// TIA Portal project "TankMixer3" (V17)

(* hardware
DEVICE "S7-1500/ET200MP station_1"  S7-1500 station
   slot 0: "Rail_0"  Rack  6ES7 590-1***0-0AA0
   slot 1: "PLC_1"  CPU 1512C-1 PN  6ES7 512-1CK00-0AB0  V2.9
      slot 3: "CPU display_1"  6ES7591-1AA00-0AA0
      slot 32768: "PROFINET interface_1"  X1
         slot 32769: "Port_1"  X1 P1
         slot 32770: "Port_2"  X1 P2
      slot 34817: "Virtual CP interface port_1"  Virtual CP interface port  Virtual CP interface port
*)

// ===== PLC "PLC_1"  CPU 1512C-1 PN =====

VAR_GLOBAL   // PLC tag table "Default tag table"
   "System_ON/OFF" AT %M0.0 : Bool;
   "Tag_1" AT %M0.1 : Bool;
   "Tag_2" AT %M0.2 : Bool;
END_VAR

TYPE "Filling_Tanks"
   STRUCT
      Inflow_Valve : Bool;
      Outflow_Valve : Bool;
      Tank_Level : Int;
      Low_Level : Bool;
      High_Level : Bool;
   END_STRUCT;
END_TYPE

TYPE "Main_Tank"
   STRUCT
      Draining_Valve : Bool;
      Tank_Level : Int;
      High_Level : Bool;
      Low_Level : Bool;
   END_STRUCT;
END_TYPE

TYPE "Valves_Control"
   STRUCT
      Start : Bool;
      Stop : Bool;
      Test : Bool;
      Reset : Bool;
      Status : Bool;
   END_STRUCT;
END_TYPE

DATA_BLOCK "Tank_Mixer_DB"   // DB1
{ S7_Optimized_Access := 'FALSE' }
VERSION : 0.1
   VAR
      Start_System : Bool;
      System_Stop : Bool;
      Manual_Selection : Bool;
      Auto_Selection : Bool;
      Auto_Mode : Bool;
      Manual_Mode : Bool;
      Mixer_Motor : Bool;
      Tank1 : "Filling_Tanks";
      Tank2 : "Filling_Tanks";
      Tank3 : "Filling_Tanks";
      Main_Tank : "Main_Tank";
      Inflow_Valve1 : "Valves_Control";
      Inflow_Valve2 : "Valves_Control";
      Inflow_Valve3 : "Valves_Control";
      Outflow_Valve1 : "Valves_Control";
      Outflow_Valve2 : "Valves_Control";
      Outflow_Valve3 : "Valves_Control";
      Draining_Valve : "Valves_Control";
   END_VAR
BEGIN
END_DATA_BLOCK

// folder: System blocks/Program resources

DATA_BLOCK "IEC_Timer_0_DB"   // DB2
{ S7_Optimized_Access := 'TRUE' }
AUTHOR : Simatic
FAMILY : IEC
NAME : IEC_TMR
VERSION : 1.0
// stored: InstanceOfName IEC_TIMER
"IEC_TIMER"
BEGIN
END_DATA_BLOCK

DATA_BLOCK "IEC_Timer_0_DB_1"   // DB3
{ S7_Optimized_Access := 'TRUE' }
AUTHOR : Simatic
FAMILY : IEC
NAME : IEC_TMR
VERSION : 1.0
// stored: InstanceOfName IEC_TIMER
"IEC_TIMER"
BEGIN
END_DATA_BLOCK

DATA_BLOCK "IEC_Timer_0_DB_2"   // DB4
{ S7_Optimized_Access := 'TRUE' }
AUTHOR : Simatic
FAMILY : IEC
NAME : IEC_TMR
VERSION : 1.0
// stored: InstanceOfName IEC_TIMER
"IEC_TIMER"
BEGIN
END_DATA_BLOCK

// folder: (top level)

ORGANIZATION_BLOCK "Main"   // OB1, LAD, ProgramCycle
TITLE = "Main Program Sweep (Cycle)"
{ S7_Optimized_Access := 'TRUE' }
VERSION : 0.1
   VAR_INPUT
      Initial_Call : Bool;   // Initial call of this OB
      Remanence : Bool;   // =True, if remanent data are available
   END_VAR
BEGIN

REGION Network 1: Auto Mode Selection
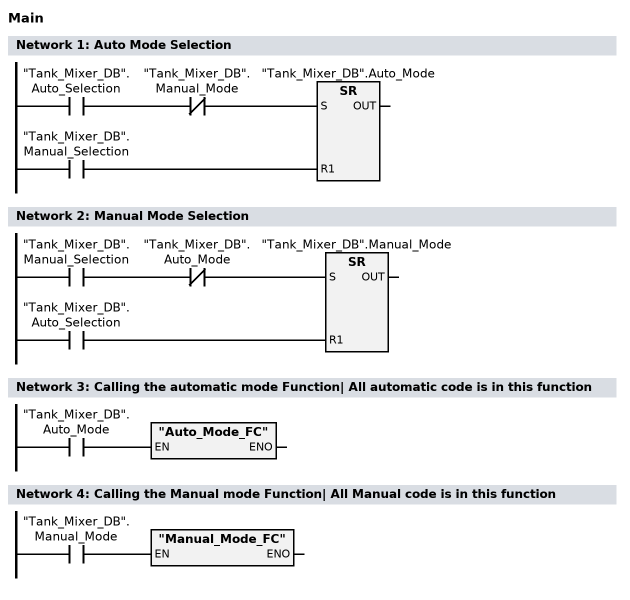
   RUNG wire#powerrail
      Contact( "Tank_Mixer_DB".Auto_Selection )
      I_Contact( "Tank_Mixer_DB".Manual_Mode )
      S_SR(operand := "Tank_Mixer_DB".Auto_Mode, r1 := wire#w1)
   END_RUNG
   RUNG wire#powerrail
      Contact( "Tank_Mixer_DB".Manual_Selection )
   END_RUNG wire#w1
   // the same network as SCL:
   IF "Tank_Mixer_DB".Auto_Selection AND NOT "Tank_Mixer_DB".Manual_Mode THEN
       "Tank_Mixer_DB".Auto_Mode := TRUE;   // SR flip-flop
   END_IF;
   IF "Tank_Mixer_DB".Manual_Selection THEN "Tank_Mixer_DB".Auto_Mode := FALSE; END_IF;
END_REGION

REGION Network 2: Manual Mode Selection
   RUNG wire#powerrail
      Contact( "Tank_Mixer_DB".Manual_Selection )
      I_Contact( "Tank_Mixer_DB".Auto_Mode )
      S_SR(operand := "Tank_Mixer_DB".Manual_Mode, r1 := wire#w1)
   END_RUNG
   RUNG wire#powerrail
      Contact( "Tank_Mixer_DB".Auto_Selection )
   END_RUNG wire#w1
   // the same network as SCL:
   IF "Tank_Mixer_DB".Manual_Selection AND NOT "Tank_Mixer_DB".Auto_Mode THEN
       "Tank_Mixer_DB".Manual_Mode := TRUE;   // SR flip-flop
   END_IF;
   IF "Tank_Mixer_DB".Auto_Selection THEN "Tank_Mixer_DB".Manual_Mode := FALSE; END_IF;
END_REGION

REGION Network 3: Calling the automatic mode Function| All automatic code is in this function
   RUNG wire#powerrail
      Contact( "Tank_Mixer_DB".Auto_Mode )
      "Auto_Mode_FC"()
   END_RUNG
   // the same network as SCL:
   IF "Tank_Mixer_DB".Auto_Mode THEN "Auto_Mode_FC"(); END_IF;
END_REGION

REGION Network 4: Calling the Manual mode Function| All Manual code is in this function
   RUNG wire#powerrail
      Contact( "Tank_Mixer_DB".Manual_Mode )
      "Manual_Mode_FC"()
   END_RUNG
   // the same network as SCL:
   IF "Tank_Mixer_DB".Manual_Mode THEN "Manual_Mode_FC"(); END_IF;
END_REGION
END_ORGANIZATION_BLOCK

// folder: Auto_Mode

FUNCTION "Auto_Mode_FC" : Void   // FC1, LAD
{ S7_Optimized_Access := 'TRUE' }
VERSION : 0.1
   VAR_TEMP   // added for the SCL form of the ladder/FBD networks
      _w1 : Bool;
   END_VAR
BEGIN

REGION Network 1
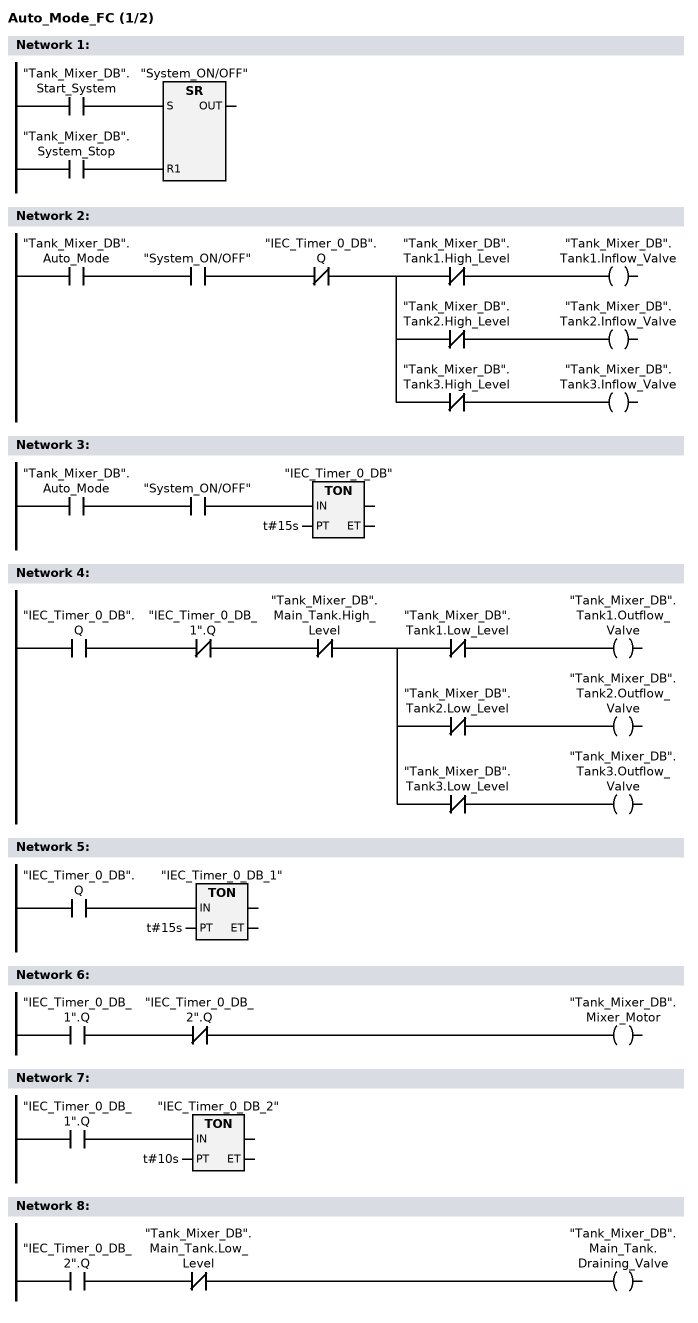
   RUNG wire#powerrail
      Contact( "Tank_Mixer_DB".Start_System )
      S_SR(operand := "System_ON/OFF", r1 := wire#w1)
   END_RUNG
   RUNG wire#powerrail
      Contact( "Tank_Mixer_DB".System_Stop )
   END_RUNG wire#w1
   // the same network as SCL:
   IF "Tank_Mixer_DB".Start_System THEN
       "System_ON/OFF" := TRUE;   // SR flip-flop
   END_IF;
   IF "Tank_Mixer_DB".System_Stop THEN "System_ON/OFF" := FALSE; END_IF;
END_REGION

REGION Network 2
   RUNG wire#powerrail
      Contact( "Tank_Mixer_DB".Auto_Mode )
      Contact( "System_ON/OFF" )
      I_Contact( "IEC_Timer_0_DB".Q )
      wire#w1
      I_Contact( "Tank_Mixer_DB".Tank1.High_Level )
      Coil( "Tank_Mixer_DB".Tank1.Inflow_Valve )
   END_RUNG
   RUNG wire#w1
      I_Contact( "Tank_Mixer_DB".Tank2.High_Level )
      Coil( "Tank_Mixer_DB".Tank2.Inflow_Valve )
   END_RUNG
   RUNG wire#w1
      I_Contact( "Tank_Mixer_DB".Tank3.High_Level )
      Coil( "Tank_Mixer_DB".Tank3.Inflow_Valve )
   END_RUNG
   // the same network as SCL:
   #_w1 := "Tank_Mixer_DB".Auto_Mode AND "System_ON/OFF" AND NOT "IEC_Timer_0_DB".Q;
   "Tank_Mixer_DB".Tank1.Inflow_Valve := #_w1 AND NOT "Tank_Mixer_DB".Tank1.High_Level;
   "Tank_Mixer_DB".Tank2.Inflow_Valve := #_w1 AND NOT "Tank_Mixer_DB".Tank2.High_Level;
   "Tank_Mixer_DB".Tank3.Inflow_Valve := #_w1 AND NOT "Tank_Mixer_DB".Tank3.High_Level;
END_REGION

REGION Network 3
   "IEC_Timer_0_DB".TON(IN := "Tank_Mixer_DB".Auto_Mode AND "System_ON/OFF", PT := t#15s);
END_REGION

REGION Network 4
   RUNG wire#powerrail
      Contact( "IEC_Timer_0_DB".Q )
      I_Contact( "IEC_Timer_0_DB_1".Q )
      I_Contact( "Tank_Mixer_DB".Main_Tank.High_Level )
      wire#w1
      I_Contact( "Tank_Mixer_DB".Tank1.Low_Level )
      Coil( "Tank_Mixer_DB".Tank1.Outflow_Valve )
   END_RUNG
   RUNG wire#w1
      I_Contact( "Tank_Mixer_DB".Tank2.Low_Level )
      Coil( "Tank_Mixer_DB".Tank2.Outflow_Valve )
   END_RUNG
   RUNG wire#w1
      I_Contact( "Tank_Mixer_DB".Tank3.Low_Level )
      Coil( "Tank_Mixer_DB".Tank3.Outflow_Valve )
   END_RUNG
   // the same network as SCL:
   #_w1 := "IEC_Timer_0_DB".Q AND NOT "IEC_Timer_0_DB_1".Q AND NOT "Tank_Mixer_DB".Main_Tank.High_Level;
   "Tank_Mixer_DB".Tank1.Outflow_Valve := #_w1 AND NOT "Tank_Mixer_DB".Tank1.Low_Level;
   "Tank_Mixer_DB".Tank2.Outflow_Valve := #_w1 AND NOT "Tank_Mixer_DB".Tank2.Low_Level;
   "Tank_Mixer_DB".Tank3.Outflow_Valve := #_w1 AND NOT "Tank_Mixer_DB".Tank3.Low_Level;
END_REGION

REGION Network 5
   "IEC_Timer_0_DB_1".TON(IN := "IEC_Timer_0_DB".Q, PT := t#15s);
END_REGION

REGION Network 6
   RUNG wire#powerrail
      Contact( "IEC_Timer_0_DB_1".Q )
      I_Contact( "IEC_Timer_0_DB_2".Q )
      Coil( "Tank_Mixer_DB".Mixer_Motor )
   END_RUNG
   // the same network as SCL:
   "Tank_Mixer_DB".Mixer_Motor := "IEC_Timer_0_DB_1".Q AND NOT "IEC_Timer_0_DB_2".Q;
END_REGION

REGION Network 7
   "IEC_Timer_0_DB_2".TON(IN := "IEC_Timer_0_DB_1".Q, PT := t#10s);
END_REGION

REGION Network 8
   RUNG wire#powerrail
      Contact( "IEC_Timer_0_DB_2".Q )
      I_Contact( "Tank_Mixer_DB".Main_Tank.Low_Level )
      Coil( "Tank_Mixer_DB".Main_Tank.Draining_Valve )
   END_RUNG
   // the same network as SCL:
   "Tank_Mixer_DB".Main_Tank.Draining_Valve := "IEC_Timer_0_DB_2".Q AND NOT "Tank_Mixer_DB".Main_Tank.Low_Level;
END_REGION

REGION Network 9
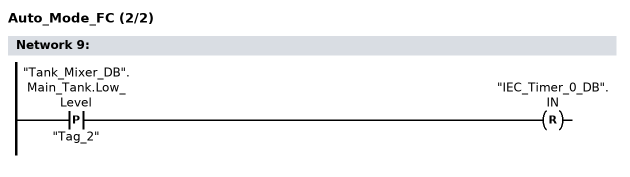
   RUNG wire#powerrail
      P_Contact(operand := "Tank_Mixer_DB".Main_Tank.Low_Level, bit := "Tag_2")
      R_Coil( "IEC_Timer_0_DB".IN )
   END_RUNG
   // the same network as SCL:
   #_w1 := "Tank_Mixer_DB".Main_Tank.Low_Level AND NOT "Tag_2";   // rising edge of "Tank_Mixer_DB".Main_Tank.Low_Level
   "Tag_2" := "Tank_Mixer_DB".Main_Tank.Low_Level;
   IF #_w1 THEN "IEC_Timer_0_DB".IN := FALSE; END_IF;
END_REGION
END_FUNCTION

FUNCTION "MainTank_Level_ControlAuto" : Void   // FC6, LAD
{ S7_Optimized_Access := 'TRUE' }
VERSION : 0.1
BEGIN

REGION Network 1
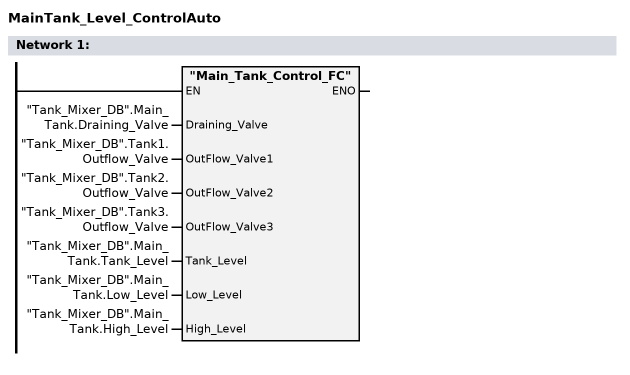
   RUNG wire#powerrail
      "Main_Tank_Control_FC"(Draining_Valve := "Tank_Mixer_DB".Main_Tank.Draining_Valve, OutFlow_Valve1 := "Tank_Mixer_DB".Tank1.Outflow_Valve, OutFlow_Valve2 := "Tank_Mixer_DB".Tank2.Outflow_Valve, OutFlow_Valve3 := "Tank_Mixer_DB".Tank3.Outflow_Valve, Tank_Level := "Tank_Mixer_DB".Main_Tank.Tank_Level, Low_Level := "Tank_Mixer_DB".Main_Tank.Low_Level, High_Level := "Tank_Mixer_DB".Main_Tank.High_Level)
   END_RUNG
   // the same network as SCL:
   "Main_Tank_Control_FC"(Draining_Valve := "Tank_Mixer_DB".Main_Tank.Draining_Valve,
                          OutFlow_Valve1 := "Tank_Mixer_DB".Tank1.Outflow_Valve,
                          OutFlow_Valve2 := "Tank_Mixer_DB".Tank2.Outflow_Valve,
                          OutFlow_Valve3 := "Tank_Mixer_DB".Tank3.Outflow_Valve,
                          Tank_Level := "Tank_Mixer_DB".Main_Tank.Tank_Level,
                          Low_Level := "Tank_Mixer_DB".Main_Tank.Low_Level,
                          High_Level := "Tank_Mixer_DB".Main_Tank.High_Level);
END_REGION
END_FUNCTION

FUNCTION "3Tanks_Level_ControlAuto" : Void   // FC9, LAD
{ S7_Optimized_Access := 'TRUE' }
VERSION : 0.1
BEGIN

REGION Network 1: TANK 1: Next 3 Ranks control the levels of the 3 tanks
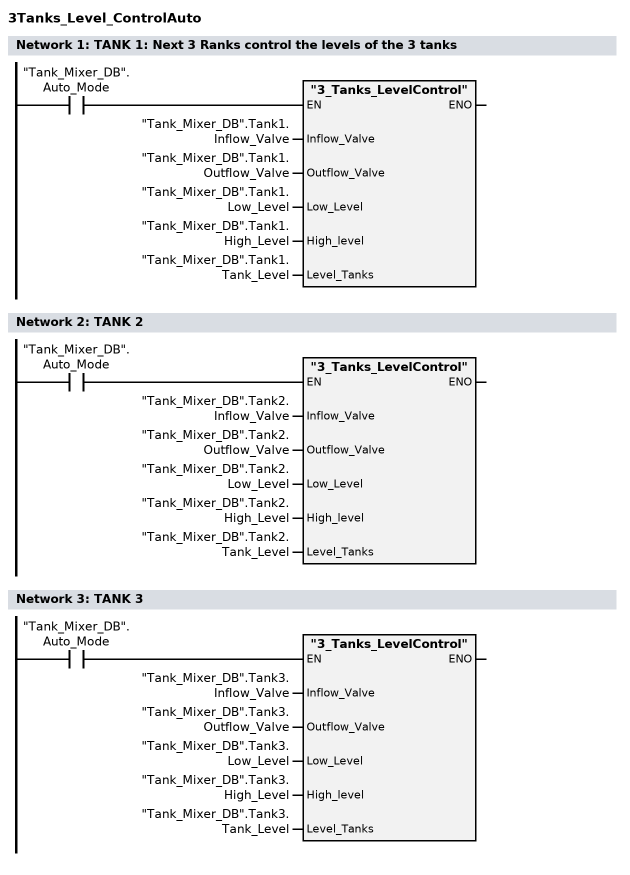
   RUNG wire#powerrail
      Contact( "Tank_Mixer_DB".Auto_Mode )
      "3_Tanks_LevelControl"(Inflow_Valve := "Tank_Mixer_DB".Tank1.Inflow_Valve, Outflow_Valve := "Tank_Mixer_DB".Tank1.Outflow_Valve, Low_Level := "Tank_Mixer_DB".Tank1.Low_Level, High_level := "Tank_Mixer_DB".Tank1.High_Level, Level_Tanks := "Tank_Mixer_DB".Tank1.Tank_Level)
   END_RUNG
   // the same network as SCL:
   IF "Tank_Mixer_DB".Auto_Mode THEN
       "3_Tanks_LevelControl"(Inflow_Valve := "Tank_Mixer_DB".Tank1.Inflow_Valve,
                              Outflow_Valve := "Tank_Mixer_DB".Tank1.Outflow_Valve,
                              Low_Level := "Tank_Mixer_DB".Tank1.Low_Level,
                              High_level := "Tank_Mixer_DB".Tank1.High_Level,
                              Level_Tanks := "Tank_Mixer_DB".Tank1.Tank_Level);
   END_IF;
END_REGION

REGION Network 2: TANK 2
   RUNG wire#powerrail
      Contact( "Tank_Mixer_DB".Auto_Mode )
      "3_Tanks_LevelControl"(Inflow_Valve := "Tank_Mixer_DB".Tank2.Inflow_Valve, Outflow_Valve := "Tank_Mixer_DB".Tank2.Outflow_Valve, Low_Level := "Tank_Mixer_DB".Tank2.Low_Level, High_level := "Tank_Mixer_DB".Tank2.High_Level, Level_Tanks := "Tank_Mixer_DB".Tank2.Tank_Level)
   END_RUNG
   // the same network as SCL:
   IF "Tank_Mixer_DB".Auto_Mode THEN
       "3_Tanks_LevelControl"(Inflow_Valve := "Tank_Mixer_DB".Tank2.Inflow_Valve,
                              Outflow_Valve := "Tank_Mixer_DB".Tank2.Outflow_Valve,
                              Low_Level := "Tank_Mixer_DB".Tank2.Low_Level,
                              High_level := "Tank_Mixer_DB".Tank2.High_Level,
                              Level_Tanks := "Tank_Mixer_DB".Tank2.Tank_Level);
   END_IF;
END_REGION

REGION Network 3: TANK 3
   RUNG wire#powerrail
      Contact( "Tank_Mixer_DB".Auto_Mode )
      "3_Tanks_LevelControl"(Inflow_Valve := "Tank_Mixer_DB".Tank3.Inflow_Valve, Outflow_Valve := "Tank_Mixer_DB".Tank3.Outflow_Valve, Low_Level := "Tank_Mixer_DB".Tank3.Low_Level, High_level := "Tank_Mixer_DB".Tank3.High_Level, Level_Tanks := "Tank_Mixer_DB".Tank3.Tank_Level)
   END_RUNG
   // the same network as SCL:
   IF "Tank_Mixer_DB".Auto_Mode THEN
       "3_Tanks_LevelControl"(Inflow_Valve := "Tank_Mixer_DB".Tank3.Inflow_Valve,
                              Outflow_Valve := "Tank_Mixer_DB".Tank3.Outflow_Valve,
                              Low_Level := "Tank_Mixer_DB".Tank3.Low_Level,
                              High_level := "Tank_Mixer_DB".Tank3.High_Level,
                              Level_Tanks := "Tank_Mixer_DB".Tank3.Tank_Level);
   END_IF;
END_REGION
END_FUNCTION

ORGANIZATION_BLOCK "Cyclic interrupt_Auto_3Tanks"   // OB30, LAD, CyclicInterrupt
{ S7_Optimized_Access := 'TRUE' }
VERSION : 0.1
   VAR_INPUT
      Initial_Call : Bool;   // Initial call of this OB
      Event_Count : Int;   // Events discarded
   END_VAR
   VAR_TEMP
      Norm_Value : Real;
   END_VAR
BEGIN

REGION Network 1
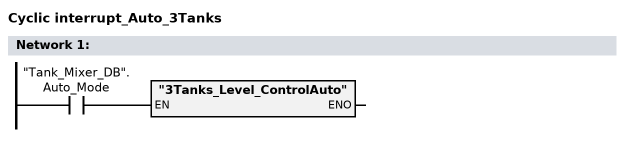
   RUNG wire#powerrail
      Contact( "Tank_Mixer_DB".Auto_Mode )
      "3Tanks_Level_ControlAuto"()
   END_RUNG
   // the same network as SCL:
   IF "Tank_Mixer_DB".Auto_Mode THEN "3Tanks_Level_ControlAuto"(); END_IF;
END_REGION
END_ORGANIZATION_BLOCK

ORGANIZATION_BLOCK "Cyclic interrupt_Auto_MainTank"   // OB32, LAD, CyclicInterrupt
{ S7_Optimized_Access := 'TRUE' }
VERSION : 0.1
   VAR_INPUT
      Initial_Call : Bool;   // Initial call of this OB
      Event_Count : Int;   // Events discarded
   END_VAR
   VAR_TEMP
      Norm_Value : Real;
   END_VAR
BEGIN

REGION Network 1
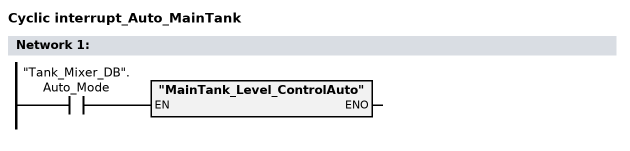
   RUNG wire#powerrail
      Contact( "Tank_Mixer_DB".Auto_Mode )
      "MainTank_Level_ControlAuto"()
   END_RUNG
   // the same network as SCL:
   IF "Tank_Mixer_DB".Auto_Mode THEN "MainTank_Level_ControlAuto"(); END_IF;
END_REGION
END_ORGANIZATION_BLOCK

// folder: Manual_Mode

FUNCTION "3Tanks_Level_ControlsManual" : Void   // FC2, LAD
{ S7_Optimized_Access := 'TRUE' }
VERSION : 0.1
BEGIN

REGION Network 1: TANK 1_LEVEL_CONTROL
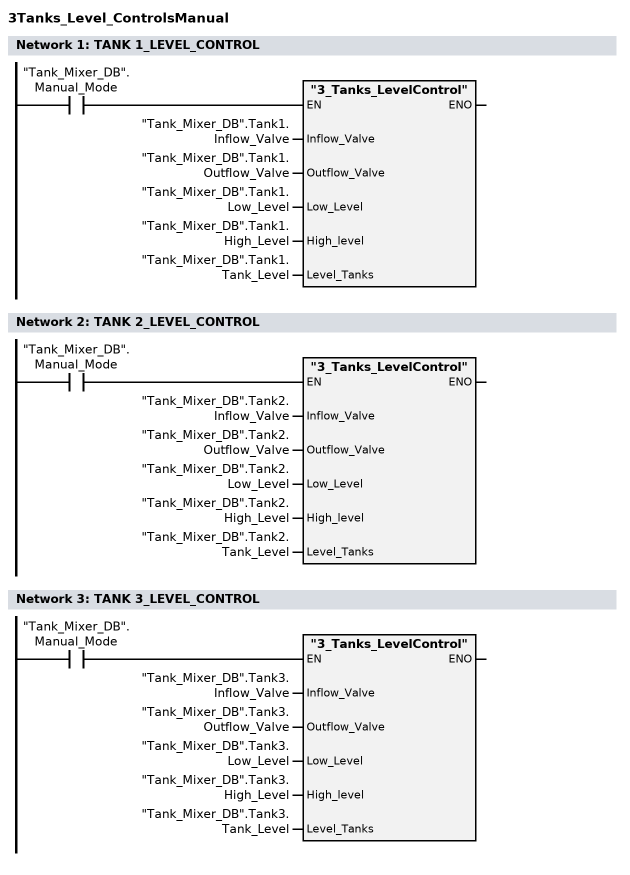
   RUNG wire#powerrail
      Contact( "Tank_Mixer_DB".Manual_Mode )
      "3_Tanks_LevelControl"(Inflow_Valve := "Tank_Mixer_DB".Tank1.Inflow_Valve, Outflow_Valve := "Tank_Mixer_DB".Tank1.Outflow_Valve, Low_Level := "Tank_Mixer_DB".Tank1.Low_Level, High_level := "Tank_Mixer_DB".Tank1.High_Level, Level_Tanks := "Tank_Mixer_DB".Tank1.Tank_Level)
   END_RUNG
   // the same network as SCL:
   IF "Tank_Mixer_DB".Manual_Mode THEN
       "3_Tanks_LevelControl"(Inflow_Valve := "Tank_Mixer_DB".Tank1.Inflow_Valve,
                              Outflow_Valve := "Tank_Mixer_DB".Tank1.Outflow_Valve,
                              Low_Level := "Tank_Mixer_DB".Tank1.Low_Level,
                              High_level := "Tank_Mixer_DB".Tank1.High_Level,
                              Level_Tanks := "Tank_Mixer_DB".Tank1.Tank_Level);
   END_IF;
END_REGION

REGION Network 2: TANK 2_LEVEL_CONTROL
   RUNG wire#powerrail
      Contact( "Tank_Mixer_DB".Manual_Mode )
      "3_Tanks_LevelControl"(Inflow_Valve := "Tank_Mixer_DB".Tank2.Inflow_Valve, Outflow_Valve := "Tank_Mixer_DB".Tank2.Outflow_Valve, Low_Level := "Tank_Mixer_DB".Tank2.Low_Level, High_level := "Tank_Mixer_DB".Tank2.High_Level, Level_Tanks := "Tank_Mixer_DB".Tank2.Tank_Level)
   END_RUNG
   // the same network as SCL:
   IF "Tank_Mixer_DB".Manual_Mode THEN
       "3_Tanks_LevelControl"(Inflow_Valve := "Tank_Mixer_DB".Tank2.Inflow_Valve,
                              Outflow_Valve := "Tank_Mixer_DB".Tank2.Outflow_Valve,
                              Low_Level := "Tank_Mixer_DB".Tank2.Low_Level,
                              High_level := "Tank_Mixer_DB".Tank2.High_Level,
                              Level_Tanks := "Tank_Mixer_DB".Tank2.Tank_Level);
   END_IF;
END_REGION

REGION Network 3: TANK 3_LEVEL_CONTROL
   RUNG wire#powerrail
      Contact( "Tank_Mixer_DB".Manual_Mode )
      "3_Tanks_LevelControl"(Inflow_Valve := "Tank_Mixer_DB".Tank3.Inflow_Valve, Outflow_Valve := "Tank_Mixer_DB".Tank3.Outflow_Valve, Low_Level := "Tank_Mixer_DB".Tank3.Low_Level, High_level := "Tank_Mixer_DB".Tank3.High_Level, Level_Tanks := "Tank_Mixer_DB".Tank3.Tank_Level)
   END_RUNG
   // the same network as SCL:
   IF "Tank_Mixer_DB".Manual_Mode THEN
       "3_Tanks_LevelControl"(Inflow_Valve := "Tank_Mixer_DB".Tank3.Inflow_Valve,
                              Outflow_Valve := "Tank_Mixer_DB".Tank3.Outflow_Valve,
                              Low_Level := "Tank_Mixer_DB".Tank3.Low_Level,
                              High_level := "Tank_Mixer_DB".Tank3.High_Level,
                              Level_Tanks := "Tank_Mixer_DB".Tank3.Tank_Level);
   END_IF;
END_REGION
END_FUNCTION

FUNCTION "Manual_Mode_FC" : Void   // FC4, LAD
{ S7_Optimized_Access := 'TRUE' }
VERSION : 0.1
BEGIN

REGION Network 1: START_SYSTEM
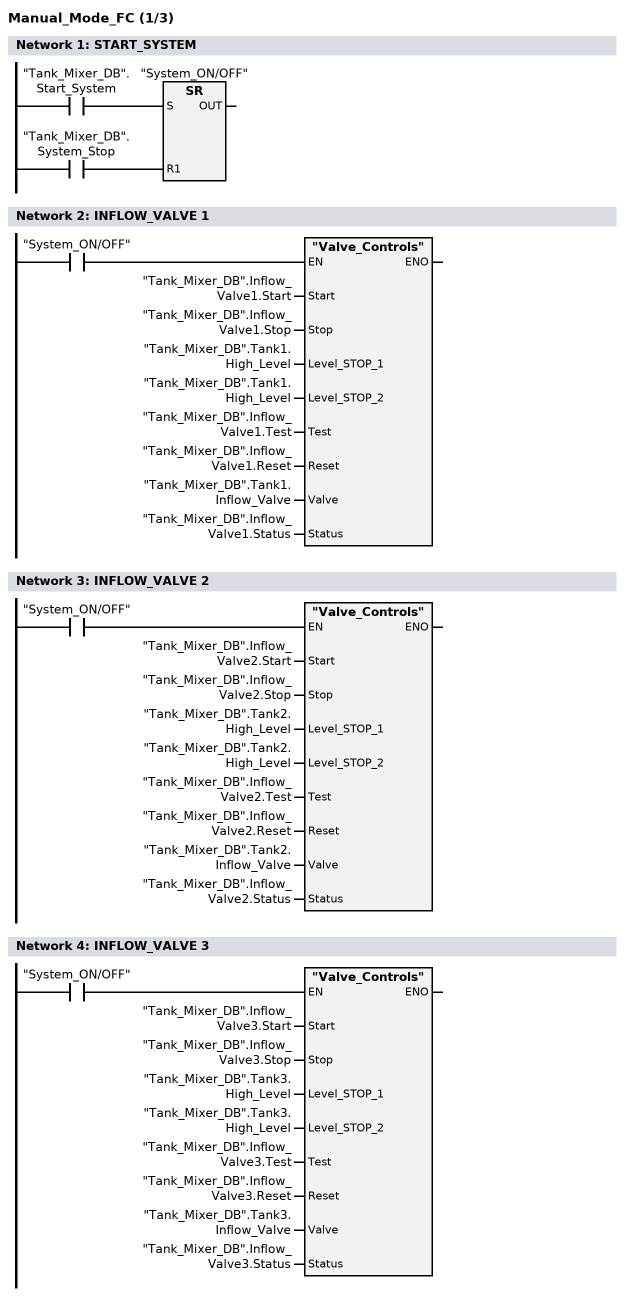
   RUNG wire#powerrail
      Contact( "Tank_Mixer_DB".Start_System )
      S_SR(operand := "System_ON/OFF", r1 := wire#w1)
   END_RUNG
   RUNG wire#powerrail
      Contact( "Tank_Mixer_DB".System_Stop )
   END_RUNG wire#w1
   // the same network as SCL:
   IF "Tank_Mixer_DB".Start_System THEN
       "System_ON/OFF" := TRUE;   // SR flip-flop
   END_IF;
   IF "Tank_Mixer_DB".System_Stop THEN "System_ON/OFF" := FALSE; END_IF;
END_REGION

REGION Network 2: INFLOW_VALVE 1
   RUNG wire#powerrail
      Contact( "System_ON/OFF" )
      "Valve_Controls"(Start := "Tank_Mixer_DB".Inflow_Valve1.Start, Stop := "Tank_Mixer_DB".Inflow_Valve1.Stop, Level_STOP_1 := "Tank_Mixer_DB".Tank1.High_Level, Level_STOP_2 := "Tank_Mixer_DB".Tank1.High_Level, Test := "Tank_Mixer_DB".Inflow_Valve1.Test, Reset := "Tank_Mixer_DB".Inflow_Valve1.Reset, Valve := "Tank_Mixer_DB".Tank1.Inflow_Valve, Status := "Tank_Mixer_DB".Inflow_Valve1.Status)
   END_RUNG
   // the same network as SCL:
   IF "System_ON/OFF" THEN
       "Valve_Controls"(Start := "Tank_Mixer_DB".Inflow_Valve1.Start,
                        Stop := "Tank_Mixer_DB".Inflow_Valve1.Stop,
                        Level_STOP_1 := "Tank_Mixer_DB".Tank1.High_Level,
                        Level_STOP_2 := "Tank_Mixer_DB".Tank1.High_Level,
                        Test := "Tank_Mixer_DB".Inflow_Valve1.Test,
                        Reset := "Tank_Mixer_DB".Inflow_Valve1.Reset,
                        Valve := "Tank_Mixer_DB".Tank1.Inflow_Valve,
                        Status := "Tank_Mixer_DB".Inflow_Valve1.Status);
   END_IF;
END_REGION

REGION Network 3: INFLOW_VALVE 2
   RUNG wire#powerrail
      Contact( "System_ON/OFF" )
      "Valve_Controls"(Start := "Tank_Mixer_DB".Inflow_Valve2.Start, Stop := "Tank_Mixer_DB".Inflow_Valve2.Stop, Level_STOP_1 := "Tank_Mixer_DB".Tank2.High_Level, Level_STOP_2 := "Tank_Mixer_DB".Tank2.High_Level, Test := "Tank_Mixer_DB".Inflow_Valve2.Test, Reset := "Tank_Mixer_DB".Inflow_Valve2.Reset, Valve := "Tank_Mixer_DB".Tank2.Inflow_Valve, Status := "Tank_Mixer_DB".Inflow_Valve2.Status)
   END_RUNG
   // the same network as SCL:
   IF "System_ON/OFF" THEN
       "Valve_Controls"(Start := "Tank_Mixer_DB".Inflow_Valve2.Start,
                        Stop := "Tank_Mixer_DB".Inflow_Valve2.Stop,
                        Level_STOP_1 := "Tank_Mixer_DB".Tank2.High_Level,
                        Level_STOP_2 := "Tank_Mixer_DB".Tank2.High_Level,
                        Test := "Tank_Mixer_DB".Inflow_Valve2.Test,
                        Reset := "Tank_Mixer_DB".Inflow_Valve2.Reset,
                        Valve := "Tank_Mixer_DB".Tank2.Inflow_Valve,
                        Status := "Tank_Mixer_DB".Inflow_Valve2.Status);
   END_IF;
END_REGION

REGION Network 4: INFLOW_VALVE 3
   RUNG wire#powerrail
      Contact( "System_ON/OFF" )
      "Valve_Controls"(Start := "Tank_Mixer_DB".Inflow_Valve3.Start, Stop := "Tank_Mixer_DB".Inflow_Valve3.Stop, Level_STOP_1 := "Tank_Mixer_DB".Tank3.High_Level, Level_STOP_2 := "Tank_Mixer_DB".Tank3.High_Level, Test := "Tank_Mixer_DB".Inflow_Valve3.Test, Reset := "Tank_Mixer_DB".Inflow_Valve3.Reset, Valve := "Tank_Mixer_DB".Tank3.Inflow_Valve, Status := "Tank_Mixer_DB".Inflow_Valve3.Status)
   END_RUNG
   // the same network as SCL:
   IF "System_ON/OFF" THEN
       "Valve_Controls"(Start := "Tank_Mixer_DB".Inflow_Valve3.Start,
                        Stop := "Tank_Mixer_DB".Inflow_Valve3.Stop,
                        Level_STOP_1 := "Tank_Mixer_DB".Tank3.High_Level,
                        Level_STOP_2 := "Tank_Mixer_DB".Tank3.High_Level,
                        Test := "Tank_Mixer_DB".Inflow_Valve3.Test,
                        Reset := "Tank_Mixer_DB".Inflow_Valve3.Reset,
                        Valve := "Tank_Mixer_DB".Tank3.Inflow_Valve,
                        Status := "Tank_Mixer_DB".Inflow_Valve3.Status);
   END_IF;
END_REGION

REGION Network 5: OUTFLOW_VALVE 1
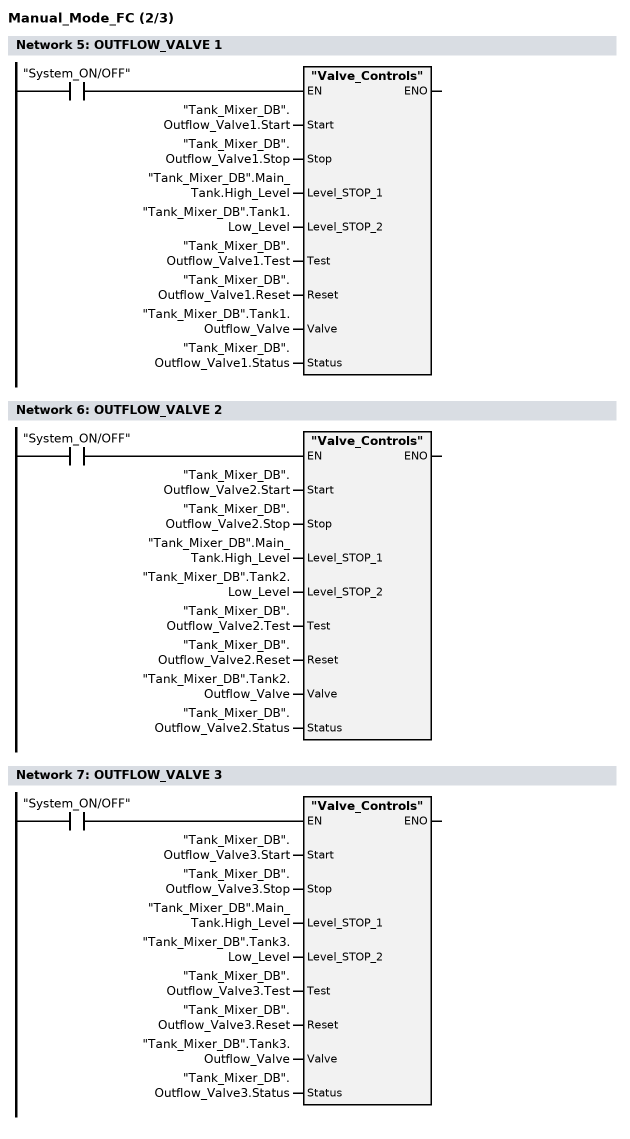
   RUNG wire#powerrail
      Contact( "System_ON/OFF" )
      "Valve_Controls"(Start := "Tank_Mixer_DB".Outflow_Valve1.Start, Stop := "Tank_Mixer_DB".Outflow_Valve1.Stop, Level_STOP_1 := "Tank_Mixer_DB".Main_Tank.High_Level, Level_STOP_2 := "Tank_Mixer_DB".Tank1.Low_Level, Test := "Tank_Mixer_DB".Outflow_Valve1.Test, Reset := "Tank_Mixer_DB".Outflow_Valve1.Reset, Valve := "Tank_Mixer_DB".Tank1.Outflow_Valve, Status := "Tank_Mixer_DB".Outflow_Valve1.Status)
   END_RUNG
   // the same network as SCL:
   IF "System_ON/OFF" THEN
       "Valve_Controls"(Start := "Tank_Mixer_DB".Outflow_Valve1.Start,
                        Stop := "Tank_Mixer_DB".Outflow_Valve1.Stop,
                        Level_STOP_1 := "Tank_Mixer_DB".Main_Tank.High_Level,
                        Level_STOP_2 := "Tank_Mixer_DB".Tank1.Low_Level,
                        Test := "Tank_Mixer_DB".Outflow_Valve1.Test,
                        Reset := "Tank_Mixer_DB".Outflow_Valve1.Reset,
                        Valve := "Tank_Mixer_DB".Tank1.Outflow_Valve,
                        Status := "Tank_Mixer_DB".Outflow_Valve1.Status);
   END_IF;
END_REGION

REGION Network 6: OUTFLOW_VALVE 2
   RUNG wire#powerrail
      Contact( "System_ON/OFF" )
      "Valve_Controls"(Start := "Tank_Mixer_DB".Outflow_Valve2.Start, Stop := "Tank_Mixer_DB".Outflow_Valve2.Stop, Level_STOP_1 := "Tank_Mixer_DB".Main_Tank.High_Level, Level_STOP_2 := "Tank_Mixer_DB".Tank2.Low_Level, Test := "Tank_Mixer_DB".Outflow_Valve2.Test, Reset := "Tank_Mixer_DB".Outflow_Valve2.Reset, Valve := "Tank_Mixer_DB".Tank2.Outflow_Valve, Status := "Tank_Mixer_DB".Outflow_Valve2.Status)
   END_RUNG
   // the same network as SCL:
   IF "System_ON/OFF" THEN
       "Valve_Controls"(Start := "Tank_Mixer_DB".Outflow_Valve2.Start,
                        Stop := "Tank_Mixer_DB".Outflow_Valve2.Stop,
                        Level_STOP_1 := "Tank_Mixer_DB".Main_Tank.High_Level,
                        Level_STOP_2 := "Tank_Mixer_DB".Tank2.Low_Level,
                        Test := "Tank_Mixer_DB".Outflow_Valve2.Test,
                        Reset := "Tank_Mixer_DB".Outflow_Valve2.Reset,
                        Valve := "Tank_Mixer_DB".Tank2.Outflow_Valve,
                        Status := "Tank_Mixer_DB".Outflow_Valve2.Status);
   END_IF;
END_REGION

REGION Network 7: OUTFLOW_VALVE 3
   RUNG wire#powerrail
      Contact( "System_ON/OFF" )
      "Valve_Controls"(Start := "Tank_Mixer_DB".Outflow_Valve3.Start, Stop := "Tank_Mixer_DB".Outflow_Valve3.Stop, Level_STOP_1 := "Tank_Mixer_DB".Main_Tank.High_Level, Level_STOP_2 := "Tank_Mixer_DB".Tank3.Low_Level, Test := "Tank_Mixer_DB".Outflow_Valve3.Test, Reset := "Tank_Mixer_DB".Outflow_Valve3.Reset, Valve := "Tank_Mixer_DB".Tank3.Outflow_Valve, Status := "Tank_Mixer_DB".Outflow_Valve3.Status)
   END_RUNG
   // the same network as SCL:
   IF "System_ON/OFF" THEN
       "Valve_Controls"(Start := "Tank_Mixer_DB".Outflow_Valve3.Start,
                        Stop := "Tank_Mixer_DB".Outflow_Valve3.Stop,
                        Level_STOP_1 := "Tank_Mixer_DB".Main_Tank.High_Level,
                        Level_STOP_2 := "Tank_Mixer_DB".Tank3.Low_Level,
                        Test := "Tank_Mixer_DB".Outflow_Valve3.Test,
                        Reset := "Tank_Mixer_DB".Outflow_Valve3.Reset,
                        Valve := "Tank_Mixer_DB".Tank3.Outflow_Valve,
                        Status := "Tank_Mixer_DB".Outflow_Valve3.Status);
   END_IF;
END_REGION

REGION Network 8: DRAINING_VALVE
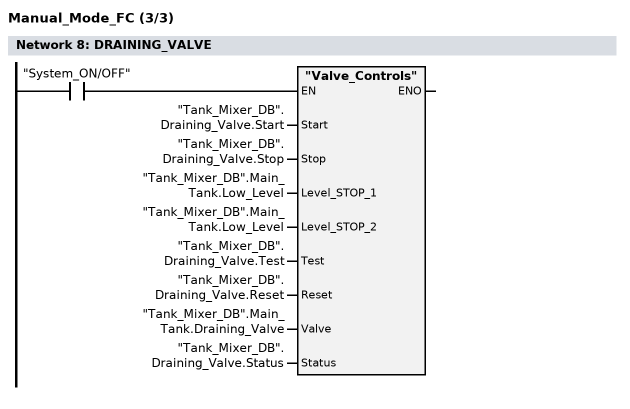
   RUNG wire#powerrail
      Contact( "System_ON/OFF" )
      "Valve_Controls"(Start := "Tank_Mixer_DB".Draining_Valve.Start, Stop := "Tank_Mixer_DB".Draining_Valve.Stop, Level_STOP_1 := "Tank_Mixer_DB".Main_Tank.Low_Level, Level_STOP_2 := "Tank_Mixer_DB".Main_Tank.Low_Level, Test := "Tank_Mixer_DB".Draining_Valve.Test, Reset := "Tank_Mixer_DB".Draining_Valve.Reset, Valve := "Tank_Mixer_DB".Main_Tank.Draining_Valve, Status := "Tank_Mixer_DB".Draining_Valve.Status)
   END_RUNG
   // the same network as SCL:
   IF "System_ON/OFF" THEN
       "Valve_Controls"(Start := "Tank_Mixer_DB".Draining_Valve.Start,
                        Stop := "Tank_Mixer_DB".Draining_Valve.Stop,
                        Level_STOP_1 := "Tank_Mixer_DB".Main_Tank.Low_Level,
                        Level_STOP_2 := "Tank_Mixer_DB".Main_Tank.Low_Level,
                        Test := "Tank_Mixer_DB".Draining_Valve.Test,
                        Reset := "Tank_Mixer_DB".Draining_Valve.Reset,
                        Valve := "Tank_Mixer_DB".Main_Tank.Draining_Valve,
                        Status := "Tank_Mixer_DB".Draining_Valve.Status);
   END_IF;
END_REGION
END_FUNCTION

FUNCTION "MainTank_Level_ControlManual" : Void   // FC7, LAD
{ S7_Optimized_Access := 'TRUE' }
VERSION : 0.1
BEGIN

REGION Network 1: MainTank_LevelSimulation
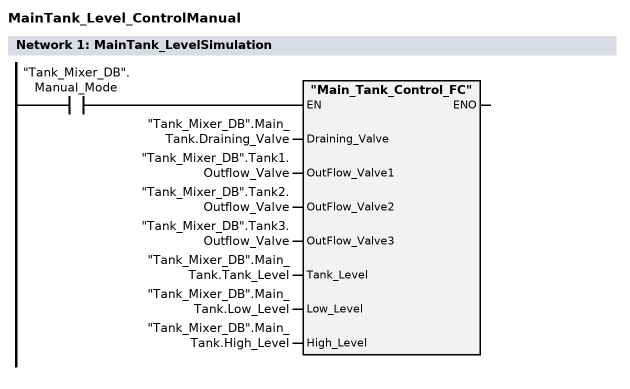
   RUNG wire#powerrail
      Contact( "Tank_Mixer_DB".Manual_Mode )
      "Main_Tank_Control_FC"(Draining_Valve := "Tank_Mixer_DB".Main_Tank.Draining_Valve, OutFlow_Valve1 := "Tank_Mixer_DB".Tank1.Outflow_Valve, OutFlow_Valve2 := "Tank_Mixer_DB".Tank2.Outflow_Valve, OutFlow_Valve3 := "Tank_Mixer_DB".Tank3.Outflow_Valve, Tank_Level := "Tank_Mixer_DB".Main_Tank.Tank_Level, Low_Level := "Tank_Mixer_DB".Main_Tank.Low_Level, High_Level := "Tank_Mixer_DB".Main_Tank.High_Level)
   END_RUNG
   // the same network as SCL:
   IF "Tank_Mixer_DB".Manual_Mode THEN
       "Main_Tank_Control_FC"(Draining_Valve := "Tank_Mixer_DB".Main_Tank.Draining_Valve,
                              OutFlow_Valve1 := "Tank_Mixer_DB".Tank1.Outflow_Valve,
                              OutFlow_Valve2 := "Tank_Mixer_DB".Tank2.Outflow_Valve,
                              OutFlow_Valve3 := "Tank_Mixer_DB".Tank3.Outflow_Valve,
                              Tank_Level := "Tank_Mixer_DB".Main_Tank.Tank_Level,
                              Low_Level := "Tank_Mixer_DB".Main_Tank.Low_Level,
                              High_Level := "Tank_Mixer_DB".Main_Tank.High_Level);
   END_IF;
END_REGION
END_FUNCTION

FUNCTION "Valve_Controls" : Void   // FC8, LAD
{ S7_Optimized_Access := 'TRUE' }
VERSION : 0.1
   VAR_INPUT
      Start : Bool;
      Stop : Bool;
      Level_STOP_1 : Bool;
      Level_STOP_2 : Bool;
      Test : Bool;
      Reset : Bool;
   END_VAR
   VAR_IN_OUT
      Valve : Bool;
      Status : Bool;
   END_VAR
BEGIN

REGION Network 1: Starting Valves and Stopping Them. RS Flip-flop
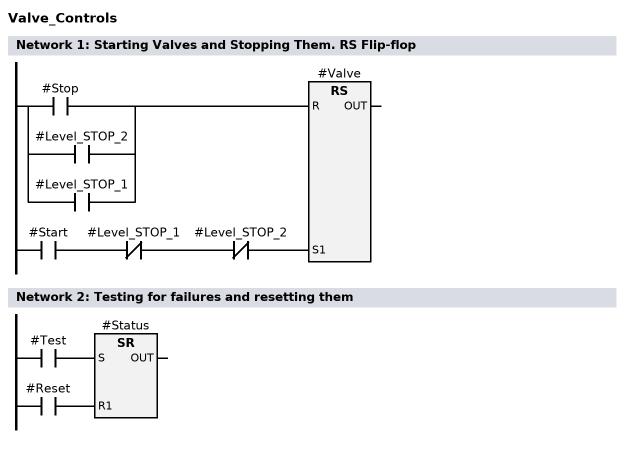
   RUNG wire#powerrail
      Contact( #Stop )
      wire#w1
      S_RS(operand := #Valve, s1 := wire#w2)
   END_RUNG
   RUNG wire#powerrail
      Contact( #Level_STOP_2 )
   END_RUNG wire#w1
   RUNG wire#powerrail
      Contact( #Level_STOP_1 )
   END_RUNG wire#w1
   RUNG wire#powerrail
      Contact( #Start )
      I_Contact( #Level_STOP_1 )
      I_Contact( #Level_STOP_2 )
   END_RUNG wire#w2
   // the same network as SCL:
   IF #Stop OR #Level_STOP_2 OR #Level_STOP_1 THEN
       #Valve := FALSE;   // RS flip-flop
   END_IF;
   IF #Start AND NOT #Level_STOP_1 AND NOT #Level_STOP_2 THEN #Valve := TRUE; END_IF;
END_REGION

REGION Network 2: Testing for failures and resetting them
   RUNG wire#powerrail
      Contact( #Test )
      S_SR(operand := #Status, r1 := wire#w1)
   END_RUNG
   RUNG wire#powerrail
      Contact( #Reset )
   END_RUNG wire#w1
   // the same network as SCL:
   IF #Test THEN
       #Status := TRUE;   // SR flip-flop
   END_IF;
   IF #Reset THEN #Status := FALSE; END_IF;
END_REGION
END_FUNCTION

ORGANIZATION_BLOCK "Cyclic interrupt_Manual_3Tanks"   // OB31, LAD, CyclicInterrupt
{ S7_Optimized_Access := 'TRUE' }
VERSION : 0.1
   VAR_INPUT
      Initial_Call : Bool;   // Initial call of this OB
      Event_Count : Int;   // Events discarded
   END_VAR
   VAR_TEMP
      Norm_Value : Real;
   END_VAR
BEGIN

REGION Network 1
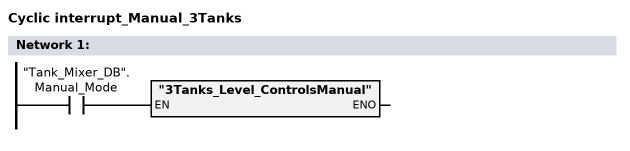
   RUNG wire#powerrail
      Contact( "Tank_Mixer_DB".Manual_Mode )
      "3Tanks_Level_ControlsManual"()
   END_RUNG
   // the same network as SCL:
   IF "Tank_Mixer_DB".Manual_Mode THEN "3Tanks_Level_ControlsManual"(); END_IF;
END_REGION
END_ORGANIZATION_BLOCK

ORGANIZATION_BLOCK "Cyclic interrupt_Manual_MainTank"   // OB33, LAD, CyclicInterrupt
{ S7_Optimized_Access := 'TRUE' }
VERSION : 0.1
   VAR_INPUT
      Initial_Call : Bool;   // Initial call of this OB
      Event_Count : Int;   // Events discarded
   END_VAR
   VAR_TEMP
      Norm_Value : Real;
   END_VAR
BEGIN

REGION Network 1
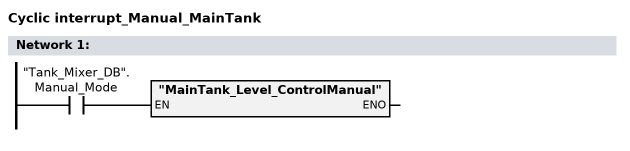
   RUNG wire#powerrail
      Contact( "Tank_Mixer_DB".Manual_Mode )
      "MainTank_Level_ControlManual"()
   END_RUNG
   // the same network as SCL:
   IF "Tank_Mixer_DB".Manual_Mode THEN "MainTank_Level_ControlManual"(); END_IF;
END_REGION
END_ORGANIZATION_BLOCK

// folder: Shared_Functions

FUNCTION "3_Tanks_LevelControl" : Void   // FC3, LAD
{ S7_Optimized_Access := 'TRUE' }
VERSION : 0.1
   VAR_INPUT
      Inflow_Valve : Bool;
      Outflow_Valve : Bool;
   END_VAR
   VAR_IN_OUT
      Low_Level : Bool;
      High_level : Bool;
      Level_Tanks : Int;
   END_VAR
BEGIN

REGION Network 1: If Inflow Valve is ON add 1 to the tank Level
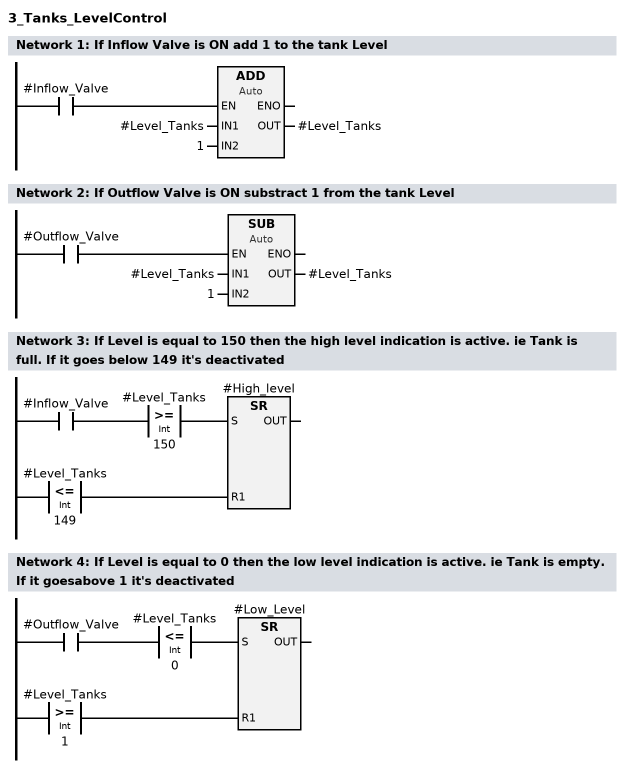
   RUNG wire#powerrail
      Contact( #Inflow_Valve )
      Add(in1 := #Level_Tanks, in2 := 1, out => #Level_Tanks)
   END_RUNG
   // the same network as SCL:
   IF #Inflow_Valve THEN #Level_Tanks := #Level_Tanks + 1; END_IF;
END_REGION

REGION Network 2: If Outflow Valve is ON substract 1 from the tank Level
   RUNG wire#powerrail
      Contact( #Outflow_Valve )
      Sub(in1 := #Level_Tanks, in2 := 1, out => #Level_Tanks)
   END_RUNG
   // the same network as SCL:
   IF #Outflow_Valve THEN #Level_Tanks := #Level_Tanks - 1; END_IF;
END_REGION

REGION Network 3: If Level is equal to 150 then the high level indication is active. ie Tank is full. If it goes below 149 it's deactivated
   RUNG wire#powerrail
      Contact( #Inflow_Valve )
      { S7_Templates := "SrcType := Int" } GE_Contact(in1 := #Level_Tanks, in2 := 150)
      S_SR(operand := #High_level, r1 := wire#w1)
   END_RUNG
   RUNG wire#powerrail
      { S7_Templates := "SrcType := Int" } LE_Contact(in1 := #Level_Tanks, in2 := 149)
   END_RUNG wire#w1
   // the same network as SCL:
   IF #Inflow_Valve AND (#Level_Tanks >= 150) THEN
       #High_level := TRUE;   // SR flip-flop
   END_IF;
   IF #Level_Tanks <= 149 THEN #High_level := FALSE; END_IF;
END_REGION

REGION Network 4: If Level is equal to 0 then the low level indication is active. ie Tank is empty. If it goesabove 1 it's deactivated
   RUNG wire#powerrail
      Contact( #Outflow_Valve )
      { S7_Templates := "SrcType := Int" } LE_Contact(in1 := #Level_Tanks, in2 := 0)
      S_SR(operand := #Low_Level, r1 := wire#w1)
   END_RUNG
   RUNG wire#powerrail
      { S7_Templates := "SrcType := Int" } GE_Contact(in1 := #Level_Tanks, in2 := 1)
   END_RUNG wire#w1
   // the same network as SCL:
   IF #Outflow_Valve AND (#Level_Tanks <= 0) THEN
       #Low_Level := TRUE;   // SR flip-flop
   END_IF;
   IF #Level_Tanks >= 1 THEN #Low_Level := FALSE; END_IF;
END_REGION
END_FUNCTION

FUNCTION "Main_Tank_Control_FC" : Void   // FC5, LAD
{ S7_Optimized_Access := 'TRUE' }
VERSION : 0.1
   VAR_INPUT
      Draining_Valve : Bool;
      OutFlow_Valve1 : Bool;
      OutFlow_Valve2 : Bool;
      OutFlow_Valve3 : Bool;
   END_VAR
   VAR_IN_OUT
      Tank_Level : Int;
      Low_Level : Bool;
      High_Level : Bool;
   END_VAR
BEGIN

REGION Network 1: If any of the 3 outflow Valves is on add one to the main tank, tank level
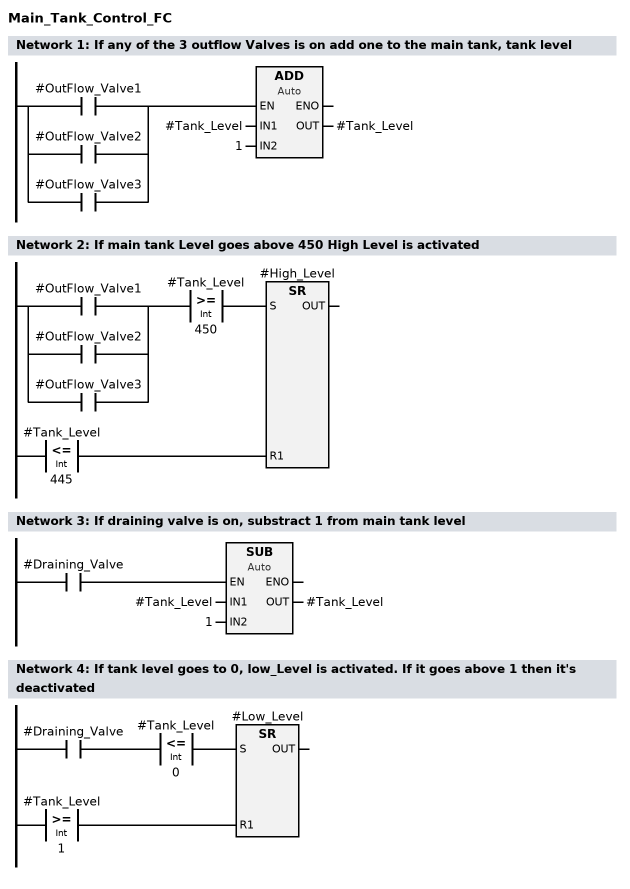
   RUNG wire#powerrail
      Contact( #OutFlow_Valve1 )
      wire#w1
      Add(in1 := #Tank_Level, in2 := 1, out => #Tank_Level)
   END_RUNG
   RUNG wire#powerrail
      Contact( #OutFlow_Valve2 )
   END_RUNG wire#w1
   RUNG wire#powerrail
      Contact( #OutFlow_Valve3 )
   END_RUNG wire#w1
   // the same network as SCL:
   IF #OutFlow_Valve1 OR #OutFlow_Valve2 OR #OutFlow_Valve3 THEN #Tank_Level := #Tank_Level + 1; END_IF;
END_REGION

REGION Network 2: If main tank Level goes above 450 High Level is activated
   RUNG wire#powerrail
      Contact( #OutFlow_Valve1 )
      wire#w1
      { S7_Templates := "SrcType := Int" } GE_Contact(in1 := #Tank_Level, in2 := 450)
      S_SR(operand := #High_Level, r1 := wire#w2)
   END_RUNG
   RUNG wire#powerrail
      Contact( #OutFlow_Valve2 )
   END_RUNG wire#w1
   RUNG wire#powerrail
      Contact( #OutFlow_Valve3 )
   END_RUNG wire#w1
   RUNG wire#powerrail
      { S7_Templates := "SrcType := Int" } LE_Contact(in1 := #Tank_Level, in2 := 445)
   END_RUNG wire#w2
   // the same network as SCL:
   IF (#OutFlow_Valve1 OR #OutFlow_Valve2 OR #OutFlow_Valve3) AND (#Tank_Level >= 450) THEN
       #High_Level := TRUE;   // SR flip-flop
   END_IF;
   IF #Tank_Level <= 445 THEN #High_Level := FALSE; END_IF;
END_REGION

REGION Network 3: If draining valve is on, substract 1 from main tank level
   RUNG wire#powerrail
      Contact( #Draining_Valve )
      Sub(in1 := #Tank_Level, in2 := 1, out => #Tank_Level)
   END_RUNG
   // the same network as SCL:
   IF #Draining_Valve THEN #Tank_Level := #Tank_Level - 1; END_IF;
END_REGION

REGION Network 4: If tank level goes to 0, low_Level is activated. If it goes above 1 then it's deactivated
   RUNG wire#powerrail
      Contact( #Draining_Valve )
      { S7_Templates := "SrcType := Int" } LE_Contact(in1 := #Tank_Level, in2 := 0)
      S_SR(operand := #Low_Level, r1 := wire#w1)
   END_RUNG
   RUNG wire#powerrail
      { S7_Templates := "SrcType := Int" } GE_Contact(in1 := #Tank_Level, in2 := 1)
   END_RUNG wire#w1
   // the same network as SCL:
   IF #Draining_Valve AND (#Tank_Level <= 0) THEN
       #Low_Level := TRUE;   // SR flip-flop
   END_IF;
   IF #Tank_Level >= 1 THEN #Low_Level := FALSE; END_IF;
END_REGION
END_FUNCTION